FUNCTION_BLOCK ABSTRACT FB_Chain EXTENDS StateMachine IMPLEMENTS I_Chain
VAR_IN_OUT
	io_fbChainController : FB_ChainController;
END_VAR
VAR_OUTPUT
	bReleaseResult : BOOL;
END_VAR
VAR
	eChainStateMachine : E_ChainStateMachine;
	uiChainNumber : UINT;
	sChainName : STRING;
	fbReleaseResult : BoolOut;
	aChainReleases : ARRAY[1..cMaxChains] OF BOOL;

	fbStepWorkerInit : FB_StepWorker;
	fbStepWorkerReady : FB_StepWorker;
	fbStepWorkerBusy : FB_StepWorker;
	fbStepWorkerWaiting : FB_StepWorker;
	fbStepWorkerError : FB_StepWorker;

	
END_VAR

SUPER^();
bReleaseResult := fbReleaseResult.getValue;

METHOD define : BOOL
VAR_INPUT
	uiChainNumber : UINT;
	sChainName    : STRING;
END_VAR
THIS^.uiChainNumber := uiChainNumber;
THIS^.sChainName := sChainName;
END_METHOD

PROPERTY getDefinition : ST_ChainDefinition
GET
getDefinition.sChainName := sChainName;
getDefinition.uiChainNumber := uiChainNumber;
END_GET
END_PROPERTY

PROPERTY getRefChainReleases : REFERENCE TO ARRAY[1..cMaxChains] OF BOOL
GET
getRefChainReleases REF= aChainReleases;
END_GET
END_PROPERTY

{warning 'Eigenschaftenimplementierung hinzufügen'}
PROPERTY getRefReleaseResult : REFERENCE TO BOOL
GET
getRefReleaseResult REF= bReleaseResult;
END_GET
END_PROPERTY

PROPERTY getReleaseResult : BoolOut
GET
getReleaseResult := fbReleaseResult;
END_GET
END_PROPERTY

END_FUNCTION_BLOCK

(* stored: Version 1.1.0.1, ProductVersion 3.1.4024.0
   POU FB_Chain: Id {61defab6-4098-4715-9800-1cf7ddffc9a5}, SpecialFunc None
   Method define: Id {6a1f9010-15d8-4362-9dd0-684cb74637ee}
   Property getDefinition: Id {dfa516b6-7b9e-48e4-b1c2-6cbfc0f5ec4f}
   Get Get: Id {9f47331d-cabd-4bee-9434-736872b919a7}
   Property getRefChainReleases: Id {8d1fbc59-ee05-4241-8382-46ea2a6dc693}
   Get Get: Id {931d6c7f-2c2d-4659-b61b-f25f84c84bbb}
   Property getRefReleaseResult: Id {9c2e1211-a1a2-406b-b645-c5646c3bc7bf}
   Get Get: Id {05877000-c74a-4b40-8f69-1ad4aeb43509}
   Property getReleaseResult: Id {89b96a0c-0e42-4023-b014-20c909692ab0}
   Get Get: Id {8216fba6-f678-4f64-97b9-1b6fff538ab8} *)
